(*			
	RafalOS
	Rafał Osajda		20.11.2025		TC 4024.66
	Moduł przygotowania danych dla Okna głównego w trybie diagnostyki
*)
FUNCTION_BLOCK FB_MCHMIPrepareDataForScreen_00_05 EXTENDS FB_MCHMIPrepareDataForScreen IMPLEMENTS ITF_MCHMIPrepareDataForScreen
VAR
	itfMachineControlHMI	: ITF_MCHMIMachineControl_HMI_PrepScr_00_05;
	refstData				: REFERENCE TO ST_MCHMIPrepareScreen_00_05;
END_VAR

(*			
	RafalOS
	Rafał Osajda		19.11.2025		TC 4024.66
	Czyści danych przy zmienia ramki po poprzedniej ramce
*)
METHOD PUBLIC ClearAfterScreen : BOOL
VAR_INPUT
END_VAR
SUPER^.ClearAfterScreen ();
END_METHOD

METHOD PUBLIC LinkDataHMI_00_05 : BOOL
VAR_INPUT
	refstData				: REFERENCE TO ST_MCHMIPrepareScreen_00_05;
END_VAR
THIS^.refstData REF= refstData;
END_METHOD

METHOD PUBLIC LinkMachineControlHMI : BOOL
VAR_INPUT
	fbMachineControlHMI	: ITF_MCHMIMachineControl_HMI_PrepScr_00_05;
END_VAR
this^.itfMachineControlHMI := fbMachineControlHMI;
END_METHOD

(*			
	RafalOS
	Rafał Osajda		14.11.2025		TC 4024.66
	Metoda przygotowywania danych dla HMI 
	W niej odbywa się odpytywanie właściego elementu przez łącznik
*)
METHOD PUBLIC PrepareDataForHMI : BOOL
VAR_INPUT
END_VAR
SUPER^.PrepareDataForHMI ();
END_METHOD

(*			
	RafalOS
	Rafał Osajda		19.11.2025		TC 4024.66
	Przygotowanie ramki pood tamke do wyświetlenia - tylko przygotowanie a nie przygotowanie danych do wyświetlenia
*)
METHOD PUBLIC PrepareForScreen : BOOL
VAR_INPUT
END_VAR
SUPER^.PrepareForScreen ();
END_METHOD

END_FUNCTION_BLOCK

(* stored: Version 1.1.0.1
   POU FB_MCHMIPrepareDataForScreen_00_05: Id {954db09e-1f6c-0c29-10b3-e817772a9a6a}, SpecialFunc None
   Folder ITF_PDFS: Id {a3e53ba1-eda8-0247-182b-33a15a71da3d}
   Method ClearAfterScreen: Id {1760cb22-cfbe-0e82-3c2a-c7a38e0700d1}
   Method LinkDataHMI_00_05: Id {e52525f6-28af-0abe-1e1c-a91e085a086b}
   Method LinkMachineControlHMI: Id {f5373edf-6147-0b1d-3f9a-1508655706f8}
   Method PrepareDataForHMI: Id {7222a4d7-c60a-088e-0812-51851dc3c64d}
   Method PrepareForScreen: Id {26ac8842-2e4b-0990-0eee-88c0373eb1da} *)
